// TIA Portal V19 export
DATA_BLOCK "PPrgArchive6"   // DB508
// stored: IsOnlyStoredInLoadMemory true, MemoryReserve 0, Namespace G
   VAR RETAIN
      PRG : Array[501..600] of "PPrg_Data";
   END_VAR
BEGIN
END_DATA_BLOCK
